KUKA KRL data list: KVP_SendPos.dat

&ACCESS RVP
&REL 4
DEFDAT KVP_SendPos PUBLIC

DECL E6POS MyPos
DECL BOOL MyBool

ENDDAT
